{attribute 'qualified_only'}
VAR_GLOBAL CONSTANT
	nChannelSize		: UDINT(1..16#FFFFFFE) := 100;
	nBaseSlotAlloc		: UDINT := 1;
END_VAR

(* stored: Version 1.1.0.1
   GVL Param: Id {257743f2-67a2-43da-bad7-f53be5f08e22}, ParameterList True *)
